SUBAPPLICATION Uebung_054 (* DigitalInput_I1-_I4 auf DigitalOutput_Q1-_Q4 *)
  (* Standard: 61499-2; Description: Copyright (c) 2023 Meisterschulen am Ostbahnhof This program and the accompanying materials are made available under the terms of the Eclipse Public License 2.0 which is available at https://www.eclipse.org/legal/epl-2.0/ SPDX-License-Identifier: EPL-2.0 *)
  (* Version 1.0, 2023-10-23, Franz Höpfinger, Meisterschulen am Ostbahnhof *)
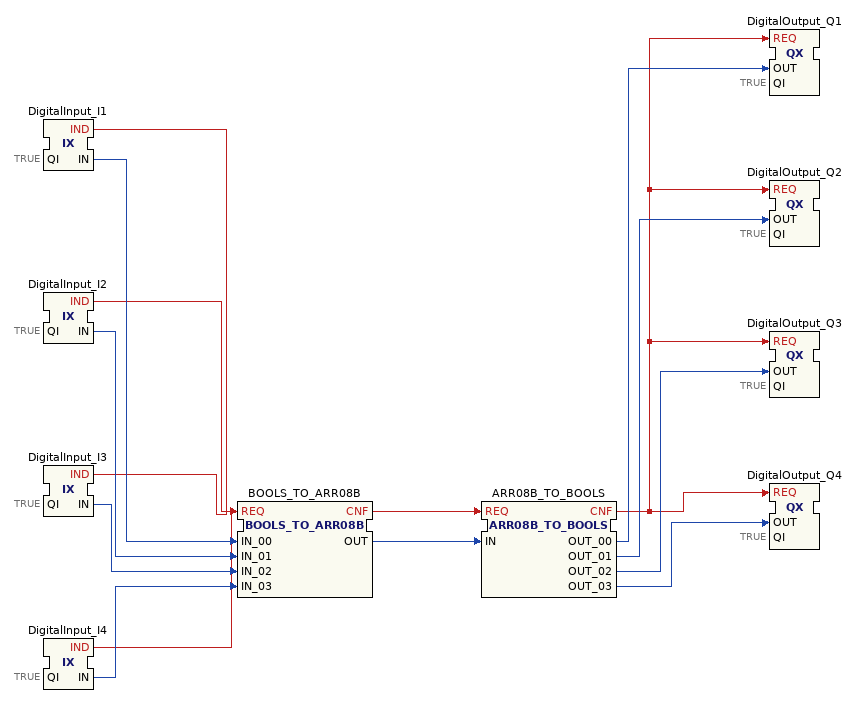
  FBS
    DigitalOutput_Q1 : QX(QI := TRUE);
    DigitalInput_I1 : IX(QI := TRUE);
    DigitalOutput_Q2 : QX(QI := TRUE);
    DigitalInput_I2 : IX(QI := TRUE);
    DigitalOutput_Q3 : QX(QI := TRUE);
    DigitalInput_I3 : IX(QI := TRUE);
    DigitalOutput_Q4 : QX(QI := TRUE);
    DigitalInput_I4 : IX(QI := TRUE);
    ARR08B_TO_BOOLS : ARR08B_TO_BOOLS;
    BOOLS_TO_ARR08B : BOOLS_TO_ARR08B;
  END_FBS
  EVENT_CONNECTIONS
    BOOLS_TO_ARR08B.CNF TO ARR08B_TO_BOOLS.REQ;
    DigitalInput_I1.IND TO BOOLS_TO_ARR08B.REQ;
    DigitalInput_I2.IND TO BOOLS_TO_ARR08B.REQ;
    DigitalInput_I3.IND TO BOOLS_TO_ARR08B.REQ;
    DigitalInput_I4.IND TO BOOLS_TO_ARR08B.REQ;
    ARR08B_TO_BOOLS.CNF TO DigitalOutput_Q1.REQ;
    ARR08B_TO_BOOLS.CNF TO DigitalOutput_Q2.REQ;
    ARR08B_TO_BOOLS.CNF TO DigitalOutput_Q3.REQ;
    ARR08B_TO_BOOLS.CNF TO DigitalOutput_Q4.REQ;
  END_CONNECTIONS
  DATA_CONNECTIONS
    BOOLS_TO_ARR08B.OUT TO ARR08B_TO_BOOLS.IN;
    DigitalInput_I1.IN TO BOOLS_TO_ARR08B.IN_00;
    DigitalInput_I2.IN TO BOOLS_TO_ARR08B.IN_01;
    DigitalInput_I3.IN TO BOOLS_TO_ARR08B.IN_02;
    DigitalInput_I4.IN TO BOOLS_TO_ARR08B.IN_03;
    ARR08B_TO_BOOLS.OUT_00 TO DigitalOutput_Q1.OUT;
    ARR08B_TO_BOOLS.OUT_01 TO DigitalOutput_Q2.OUT;
    ARR08B_TO_BOOLS.OUT_02 TO DigitalOutput_Q3.OUT;
    ARR08B_TO_BOOLS.OUT_03 TO DigitalOutput_Q4.OUT;
  END_CONNECTIONS
END_SUBAPPLICATION
